# EPICS autosave request: iocBoot/sioc-esb-stn0/stnCtrl.req
file ../stnCtrlCommon.req P=$(P)
